PROGRAM MAIN
VAR
	bInit: BOOL := TRUE;
	fbSocketCloseAll: FB_SocketCloseAll; 
	bSocketCloseError: BOOL;
	nSocketCloseError: UDINT;
	
	fbTcpClient1					: FB_TCPClient;
		sClient1SendData			: STRING(255);
		nServer1Port				: UDINT 				:= 12000;
		sServer1Host				: T_IPv4Addr 			:= '';
		bStartClient1Communication	: BOOL 					:= TRUE;
		tClient1CycleTime			: TIME 					:= T#0.5S;
		bClient1SendTrigger			: BOOL;
		bClient1Connected			: BOOL;
		sClient1ReceivedData		: STRING(255);
		bClient1Busy				: BOOL;
		bClientError1				: BOOL;
		nClient1ErrorID1			: UDINT;		
		
	fbTcpEchoServer1				: FB_TCPServer;
		sServerReceivedData			: STRING(255);
		bStartServer1Communication	: BOOL 					:= TRUE;
		bServer1Connected			: BOOL;
		sServerData					: STRING(255);
		bServer1Busy				: BOOL;
		bServer1Error				: BOOL;
		nServer1ErrorID				: UDINT;
	
	bAutogenerateData				: BOOL 					:= TRUE;
	fbTimer1						: TON;
	sBufferData						: STRING 				:= 'TestString No.';
	nCnt							: UDINT;
	
// Optional second Client and Server
(*	fbTcpClient2					: FB_TCPClient;
		sClient2SendData			: STRING(255)			:= 'TestString123';
		sClient2ReceivedData		: STRING(255);			
	fbTcpServer2					: FB_TCPServer;
		sServer2Data				: STRING(255); *)
	CYCLES: DINT;
END_VAR

CYCLES:=CYCLES+1;


IF bInit THEN 				// Init Step to close all sockets after login PLC with  downlaod
	fbSocketCloseAll(
		sSrvNetId:= '', 
		bExecute:= TRUE, 
		tTimeout:= T#3S, 
		bBusy=> , 
		bError=> bSocketCloseError, 
		nErrId=> nSocketCloseError);
	IF NOT (fbSocketCloseAll.bBusy OR fbSocketCloseAll.bError) THEN
		bInit := FALSE;
		fbSocketCloseAll(bExecute:= FALSE);
	END_IF
ELSE
	
	fbTcpClient1(
		nRemotePort:= nServer1Port, 								// Server port
		sRemoteHost:= sServer1Host, 								// Server IP (empty for local communication)
		bStartCommunication:= bStartClient1Communication, 			// Start communication, when FALSE, connection is closed
		sSendData:= sClient1SendData, 								// Data that are sent to the server
		tCycleTimeSend:= (*tClient1CycleTime*), 						// Time for cyclic sending
		bSendTrigger:= fbTimer1.Q,							// Trigger to send one telegramm manually 
		bConnected => bClient1Connected,							// Switches to TRUE when Client is connected to a server
		sReceivedData=> sClient1ReceivedData,						// Data that are received
		bBusy=> bClient1Busy, 
		bError=> bClientError1, 
		nErrorID=> nClient1ErrorID1, ); 
	
	IF bAutogenerateData AND bClient1Connected THEN
		fbTimer1(IN:= NOT fbTimer1.Q, PT:= tClient1CycleTime, Q=> , ET=> );
		IF fbTimer1.Q  THEN
			sClient1SendData := Concat(sBufferData, UDINT_TO_STRING(nCnt));
			nCnt := nCnt + 1;
		END_IF
	END_IF 
		
	fbTcpEchoServer1(
		sLocalHost:= '', 											// Server IP Adress
		nLocalPort:= nServer1Port, 									// Server port
		bStartCommunication:= bStartServer1Communication, 			// Allow Client-connection or close connection
		bConnected => bServer1Connected,							// Client connection is valid
		sSendData => sServerData,
		bBusy=> bServer1Busy, 
		bError=> bServer1Error, 
		nErrorID=> nServer1ErrorID);
	
	// Optional second Client and Server
	
(*	fbTcpClient2(
		sRemoteHost:= '', 
		nRemotePort:= 12001, 
		sSendData:= sClient2SendData, 
		bStartCommunication:= TRUE, 
		tCycleTimeSend:= T#2S, 
		bSendTrigger:= ,
		bConnected => , 
		sReceivedData=> sClient2ReceivedData, 
		nErrorID=> , 
		bError=> , 
		bBusy=> );
		
	fbTcpServer2(
		sLocalHost:= '', 
		nLocalPort:= 12001, 
		bStartCommunication:= TRUE, 
		sSendData => sServer2Data, 
		bBusy=> , 
		bError=> , 
		nErrorID=> ); *)
END_IF

END_PROGRAM

(* stored: Version 1.1.0.1, ProductVersion 3.1.4024.6
   POU MAIN: Id {572507de-a44a-4a7e-b7eb-52f2373576ea}, SpecialFunc None *)
